// Sets the boolean value to false if it is true and returns true if it was true before being set.
FUNCTION F_ResetOnTrue : BOOL // Whether the value was true before resetting.
VAR_INPUT
	bValue : REFERENCE TO BOOL; // Boolean value to reset.
END_VAR

IF bValue THEN bValue := FALSE; F_ResetOnTrue := TRUE; END_IF

END_FUNCTION

(* stored: Version 1.1.0.1
   POU F_ResetOnTrue: Id {13e4275b-f9c3-0091-3001-b4112664bcdc}, SpecialFunc None *)
